Staubli VAL3: Control_AxisPar.pgx

public program Control_AxisPar(num& x_nPos, num& x_nSpeed, num& x_nPrecent, num& x_nJogSpeed, bool x_bTraj)
  local string l_sItem[6]
  local num l_nNum
  local num l_nKey
  local num l_nData[6]
  local num l_nSelectIndex
begin
  //为LasMAN3.7进行配置
  //修改点位的参数


  //通过局部变量来实现内部存储


  l_nData[0]=x_nPos
  l_nData[1]=x_nSpeed
  l_nData[2]=x_nPrecent
  l_nData[3]=x_nJogSpeed

  l_sItem[0]="位置mm   :"+toString(".3",l_nData[0])
  l_sItem[1]="速度m/min:"+toString(".3",l_nData[1])
  l_sItem[2]="比例分度 :"+toString(".3",l_nData[2])
  l_sItem[3]="点动速度 :"+toString(".3",l_nData[3])
  call Control_BottomS(",,,,,,取消,确定")

  call Control_PanelXY(8,0,17,4)
  call Control_Panel("参数")
  call Control_List(l_sItem,l_nSelectIndex)


  //按键响应
  while true
    l_nKey=getKey()

    switch l_nKey
      case 261
        l_nSelectIndex=max(0,l_nSelectIndex-1)
      break

      case 266
        if x_bTraj
          l_nSelectIndex=min(1,l_nSelectIndex+1)
        else
           l_nSelectIndex=min(3,l_nSelectIndex+1)
        endIf

      break

      case 278

        x_nPos=l_nData[0]
        x_nSpeed=l_nData[1]
        x_nPrecent=l_nData[2]
        x_nJogSpeed=l_nData[3]
        cls()
        return
      break


      case 277,255
        cls()
        return
      break



      case 270

        call Float_Edit(l_nData[l_nSelectIndex],nPanelLTopX+11,l_nSelectIndex+nPanelLTopY+1)


        l_nData[l_nSelectIndex]=max(0,l_nData[l_nSelectIndex])
        l_nData[3]=min(100,max(0,l_nData[3]))
      break

    endSwitch

    if l_nKey!=-1
      l_sItem[0]="位置mm   :"+toString(".3",l_nData[0])
      l_sItem[1]="速度m/min:"+toString(".3",l_nData[1])
      l_sItem[2]="比例分度 :"+toString(".3",l_nData[2])
      l_sItem[3]="点动速度 :"+toString(".3",l_nData[3])
      call Control_List(l_sItem,l_nSelectIndex)

    endIf






  endWhile

end
